// Block: Rollformer_PERS

DATA_BLOCK Rollformer_PERS
VERSION : 0.1
   NON_RETAIN
   VAR
      PersistentValues : udt_Rollformer_Pers;
   END_VAR

BEGIN
   // No initialization required
END_DATA_BLOCK
